// TIA Portal V21 export
FUNCTION "FC_Conveyor_entry" : Void   // FC2, LAD
TITLE = Control de Cinta Principal
{ S7_Optimized_Access := 'TRUE' }
// stored: SetENOAutomatically false
   VAR_INPUT
      Emergencia : Bool;
      "Sistema en marcha" : Bool;
      Clasificando : Bool;
      "Pallet sensor" : Bool;
   END_VAR
   VAR_OUTPUT
      "Conveyor entry" : Bool;
   END_VAR
BEGIN

REGION Network 1: Activacion/Descativacion de cinta principal
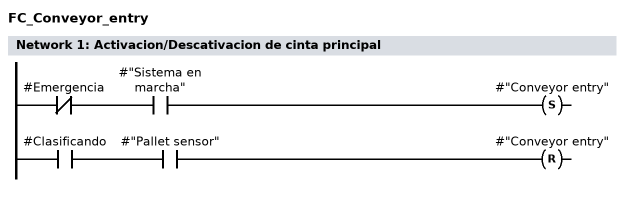
   RUNG wire#powerrail
      I_Contact( #Emergencia )
      Contact( #"Sistema en marcha" )
      S_Coil( #"Conveyor entry" )
   END_RUNG
   RUNG wire#powerrail
      Contact( #Clasificando )
      Contact( #"Pallet sensor" )
      R_Coil( #"Conveyor entry" )
   END_RUNG
   // the same network as SCL:
   IF NOT #Emergencia AND #"Sistema en marcha" THEN #"Conveyor entry" := TRUE; END_IF;
   IF #Clasificando AND #"Pallet sensor" THEN #"Conveyor entry" := FALSE; END_IF;
END_REGION
END_FUNCTION
